FUNCTION_BLOCK FB_MovingAverage
VAR_OUTPUT
	ready : BOOL;
	value : REAL;
END_VAR
VAR
    sum           : REAL;
    count         : UDINT;
    running       : BOOL;
    elapsedTime   : TIME;
	
	addToSum		: BOOL;
	elapsedSecond	: INT;
	valueArray		: ARRAY[1..999] OF REAL;
	i				: INT;
	
    intervalTime : TIME;
END_VAR

METHOD reset : BOOL
VAR_INPUT
END_VAR

value := 0;
ready := FALSE;
sum := 0;
count := 0;
running := FALSE;
elapsedTime := T#0S;
elapsedSecond := 0;
FOR i := 1 TO 999 DO
	valueArray[i] := 0;
END_FOR
END_METHOD

METHOD startCalculation : BOOL
VAR_INPUT
    start : BOOL;
    measurement : REAL;
    windowS : INT;
	intervalS : INT;
    dtime : TIME;  
	excludeUntilReady : BOOL;
END_VAR

// If window is 0, return immediately
IF windowS = 0 THEN
	RETURN;
END_IF

// Start edge
IF start AND NOT running THEN
    running := TRUE;
END_IF

IF running THEN
	elapsedTime := elapsedTime + dtime;
	intervalTime := intervalTime + dtime;
	
	// Every second, calculate new mean value and shift values forward
	IF ready THEN
		IF (TIME_TO_INT(intervalTime))/1000 >= intervalS THEN
			addToSum := TRUE;
			elapsedSecond := elapsedSecond + 1;
			FOR i := 1 TO windowS DO
				sum := sum + valueArray[i];
			END_FOR
			value := sum/windowS;
			// Shift values
			FOR i := 1 TO windowS - 1 DO
				valueArray[i] := valueArray[i + 1];
			END_FOR
			valueArray[windowS] := measurement;
			intervalTime := T#0S;
			sum := 0;
		END_IF
	ELSE
		IF (TIME_TO_INT(intervalTime))/1000 >= intervalS THEN
			elapsedSecond := elapsedSecond + 1;
			valueArray[elapsedSecond] := measurement;
			intervalTime := T#0S;
			IF NOT excludeUntilReady THEN
				FOR i := 1 TO elapsedSecond DO
					sum := sum + valueArray[i];
				END_FOR
				value := sum / elapsedSecond;
				sum := 0;
			ELSE
				value := 0;
			END_IF
		END_IF
	END_IF
	
	// After initial interval passed, start calculating the value
	IF elapsedTime >= INT_TO_TIME(windowS*1000) THEN
		startCalculation := TRUE;
		ready := TRUE;
	END_IF
	
END_IF
END_METHOD

END_FUNCTION_BLOCK

(* stored: Version 1.1.0.1, ProductVersion 3.1.4024.9
   POU FB_MovingAverage: Id {b07b32d7-af39-4b0c-93fd-b05517eb8080}, SpecialFunc None
   Method reset: Id {f6bdfb4c-6b5e-41a6-9b7e-81def0d9780d}
   Method startCalculation: Id {2a07f0e2-d431-4142-bbf5-9da0485c176e} *)
